PROGRAM PRG_UpdateGasSupply
VAR
	evtGasSupplyStart		: DetectEvent;
	evtGasSupplyStop		: DetectEvent;
END_VAR

gasSupplyPressureBar := INT_TO_REAL(gasSupplyPressureRaw)*gasSupplyPressureSensorCalibration.scaleFactor + gasSupplyPressureSensorCalibration.offset;


(* button events *)
evtGasSupplyStart(newSignalValue := gasSupplyStart);
evtGasSupplyStop(newSignalValue := gasSupplyStop);

IF evtGasSupplyStart.eventDetected = TASTEVT_PositiveEdge THEN
	gasSupplyStart := FALSE;
	gasSupplyRunning := TRUE;
END_IF

IF evtGasSupplyStop.eventDetected = TASTEVT_PositiveEdge THEN
	gasSupplyStop := FALSE;
	gasSupplyRunning := FALSE;
END_IF


IF gasSupplyRunning THEN
	IF gasSupplyPressureBar > gasSupplyPressureSetBar + 0.1 THEN
		gasSupplyValve := FALSE;
	END_IF
	
	IF gasSupplyPressureBar < gasSupplyPressureSetBar - 0.1 THEN
		gasSupplyValve := TRUE;
	END_IF
 
END_IF

END_PROGRAM

(* stored: Version 1.1.0.1, ProductVersion 3.1.4022.7
   POU PRG_UpdateGasSupply: Id {2d8e01c2-0455-4c4f-acd8-286721cc7426}, SpecialFunc None *)
